FUNCTION_BLOCK FB_ModbusRTU
VAR_INPUT
	

END_VAR
VAR_OUTPUT
END_VAR
VAR
    
 ModbusMaster   :   ModbusRtuMaster_PcCOM; 
 bExecute       : BOOL;
 bBusy          : BOOL;
 bError         : BOOL;
 nBytesRead         : UINT;
 nModbusRegister      : ARRAY [1..24] OF WORD;
 eError         : MODBUS_ERRORS;
   
// WriteModbusMaster  :   ModbusRtuMaster_PcCOM;

 bWriteExecute  : BOOL;
(* bWriteBusy     : BOOL;
 bWriteError    : BOOL; *)

 //eWriteError    : MODBUS_ERRORS;
 
 stSpindleIO	: ST_SpindleFunctions;
	
// Drive Control Command

bStop				: BOOL;
bRunEnable			: BOOL;
bDecelRamp1			: BOOL;
bDecelRamp2			: BOOL;
bFaultReset			: BOOL;
bCoastStopRequest	: BOOL;

// SpeedRef
rSpeedRefSetpoint	: REAL;
//Accel/Decel Time
rAccel_Decel		: REAL;

// Spindle Status

nErrorCode              : BYTE;
bDriveStopped           : BOOL;
bDriveRunning           : BOOL;
bDriveTripped           : BOOL;
rOutputFrequency        : REAL;
rOutputCurrent			: REAL;
nDigitalInputSts		: WORD;
nAnalogInput1			: WORD;
nAnalogInput2			: WORD;
rSpeedRefValue			: REAL;
rDCBusVoltage			: REAL;
rDriveTemp				: REAL;


END_VAR

M_SpindleControlMapping();
M_ModbusMapping();

// Read/Write Modbus commands through PC COM Serial Port
    ModbusMaster(
                        UnitID:= 1, 
                        Quantity:= 24,
                        MBAddr:= 1, 
                        cbLength:= SIZEOF(nModbusRegister) , 
                        pMemoryAddr:= ADR(nModbusRegister), 
                        Execute:= (bExecute AND NOT bWriteExecute) OR (bWriteExecute AND NOT bExecute), 
                        Timeout:= T#5S, 
                        BUSY=> bBusy, 
                        Error=> bError, 
                        ErrorId=> eError , 
                        cbRead=> nBytesRead);
                        
(*    WriteModbusMaster(
                        UnitID:= 1, 
                        Quantity:= 4, 
                        MBAddr:= 1, 
                        cbLength:= SIZEOF(nModbusRegister) , 
                        pMemoryAddr:= ADR(nModbusRegister), 
                        Execute:= bWriteExecute AND NOT bReadExecute, 
                        Timeout:= T#5S, 
                        BUSY=> bWriteBusy, 
                        Error=> bWriteError, 
                        ErrorId=> eWriteError, 
                        cbRead=> );   *)
                     
IF  bExecute THEN                          
                                                       
    ModbusMaster.ReadRegs();
  
END_IF

IF bWriteExecute THEN   
              
    ModbusMaster.WriteRegs();
  
END_IF                  

// insert text here

METHOD M_ModbusMapping : BOOL
VAR_INPUT
END_VAR
IF bExecute THEN

    stSpindleIO.ReadDriveControlCommand	:= nModbusRegister[1];
    stSpindleIO.ReadSpeedRefSetpoint	:= WORD_TO_REAL(nModbusRegister[2]);
    stSpindleIO.ReadAccel_Decel			:= WORD_TO_REAL(nModbusRegister[4]);

ELSIF bWriteExecute THEN
    
    nModbusRegister[1]                  := stSpindleIO.SetDriveControlCommand;
    nModbusRegister[2]                  :=  REAL_TO_WORD(stSpindleIO.SetSpeedRefSetpoint);
    nModbusRegister[4]                  := REAL_TO_WORD(stSpindleIO.SetAccel_Decel);

END_IF


stSpindleIO.ErrorCode.0			:=  nModbusRegister[6].0;
stSpindleIO.ErrorCode.1			:=  nModbusRegister[6].1;
stSpindleIO.ErrorCode.2			:=  nModbusRegister[6].2;
stSpindleIO.ErrorCode.3			:=  nModbusRegister[6].3;
stSpindleIO.ErrorCode.4			:=  nModbusRegister[6].4;
stSpindleIO.ErrorCode.5			:=  nModbusRegister[6].5;
stSpindleIO.ErrorCode.6			:=  nModbusRegister[6].6;
stSpindleIO.ErrorCode.7			:=  nModbusRegister[6].7;	            //	: BYTE;

stSpindleIO.DriveStatus.0		:= nModbusRegister[6].8; 	            //	: BYTE;
stSpindleIO.DriveStatus.1		:= nModbusRegister[6].9; 	            //	: BYTE;
stSpindleIO.DriveStatus.2		:= nModbusRegister[6].10; 	            //	: BYTE;
stSpindleIO.DriveStatus.3		:= nModbusRegister[6].11; 	            //	: BYTE;
stSpindleIO.DriveStatus.4		:= nModbusRegister[6].12; 	            //	: BYTE;
stSpindleIO.DriveStatus.5		:= nModbusRegister[6].13; 	            //	: BYTE;
stSpindleIO.DriveStatus.6		:= nModbusRegister[6].14; 	            //	: BYTE;
stSpindleIO.DriveStatus.7		:= nModbusRegister[6].15; 	            //	: BYTE;

stSpindleIO.OutputFreq			:= WORD_TO_REAL(nModbusRegister[7]);	//	: REAL;
stSpindleIO.OutputCurrent		:= WORD_TO_REAL(nModbusRegister[8]);	//	: REAL;
stSpindleIO.DigitalInputSts		:= nModbusRegister[11];	                //	: INT;
stSpindleIO.AnalogIn1			:= nModbusRegister[20];	                //	: INT;
stSpindleIO.AnalogIn2			:= nModbusRegister[21];	                //	: INT;
stSpindleIO.SpeedRefValue		:= WORD_TO_REAL(nModbusRegister[22]);	//	: REAL;
stSpindleIO.DCBusVoltage		:= WORD_TO_REAL(nModbusRegister[23]);	//	: REAL;
stSpindleIO.DriveTemp			:= WORD_TO_REAL(nModbusRegister[24]);	//	: REAL;
END_METHOD

METHOD M_SpindleControlMapping : BOOL
VAR_INPUT

END_VAR

VAR
END_VAR
//Read/Write Bits

// Stop/Run Enable

IF bStop THEN

	stSpindleIO.ReadDriveControlCommand.0 := FALSE;
	
ELSIF bRunEnable THEN
		
	stSpindleIO.ReadDriveControlCommand.0 := TRUE;

END_IF

// Decel Ramps

IF bDecelRamp1 THEN
	
	stSpindleIO.ReadDriveControlCommand.1 := FALSE;

ELSIF bDecelRamp2 THEN
	
	stSpindleIO.ReadDriveControlCommand.1 := TRUE;
	
END_IF;


stSpindleIO.ReadDriveControlCommand.2 := bFaultReset;
stSpindleIO.ReadDriveControlCommand.2 := bCoastStopRequest;

stSpindleIO.ReadSpeedRefSetpoint := rSpeedRefSetpoint;
stSpindleIO.ReadAccel_Decel:= rAccel_Decel;

// Read Only Bits

nErrorCode :=    stSpindleIO.ErrorCode;
bDriveStopped	:= stSpindleIO.DriveStatus.0;
bDriveRunning	:= stSpindleIO.DriveStatus.1;
bDriveTripped	:= stSpindleIO.DriveStatus.2;

rOutputFrequency	:= stSpindleIO.OutputFreq;
rOutputCurrent		:= stSpindleIO.OutputCurrent;
nDigitalInputSts	:= stSpindleIO.DigitalInputSts;
nAnalogInput1		:= stSpindleIO.AnalogIn1;
nAnalogInput2		:= stSpindleIO.AnalogIn2;
rSpeedRefValue		:= stSpindleIO.SpeedRefValue;
rDCBusVoltage		:= stSpindleIO.DCBusVoltage;
rDriveTemp			:= stSpindleIO.DriveTemp;
END_METHOD

END_FUNCTION_BLOCK

(* stored: Version 1.1.0.1, ProductVersion 3.1.4024.9
   POU FB_ModbusRTU: Id {d33eb993-f1a5-484e-9d4d-ae7861108719}, SpecialFunc None
   Method M_ModbusMapping: Id {83d865f8-d7ae-49d7-a6f4-fcb7ec40a615}
   Method M_SpindleControlMapping: Id {2f07773b-6003-410f-852f-7cd237e180e1} *)
